// Main parameters for the library.
{attribute 'qualified_only'}
VAR_GLOBAL CONSTANT
	ERROR_MESSAGE_SIZE : __UXINT := 255; // String length of an error message.
END_VAR

(* stored: Version 1.1.0.1
   GVL PARAM_Constants: Id {3dd45391-78be-041d-2dd3-bde973a9696a}, ParameterList True *)
